INTERFACE I_CloseCommand

METHOD Close
END_METHOD

PROPERTY IsClosed : Bool
GET
END_GET
END_PROPERTY

END_INTERFACE

(* stored: Version 1.1.0.1, ProductVersion 3.1.4024.11
   Itf I_CloseCommand: Id {e1c2225f-c2c0-4c87-b625-922156b50961}
   Method Close: Id {edc8b81a-462d-44c4-942f-777aaaf61946}
   Property IsClosed: Id {1c576359-fd7f-4f41-9bcc-e0c73d25517e}
   Get Get: Id {f9770f1f-1b46-42ab-bb94-568e89830f63} *)
